Staubli VAL3: onStart.pgx

program onStart()
  local num i
begin
  // logMsg
  logMsg("[KERNEL] INTERFACE:PAGE Edit trajectory")
  // disable the filter
  if saveData:mode<2
    saveData:sTrajFilter=""
  endIf
  // check it
  if saveData:sTrajType[nType]!=saveData:sTrajTypeUsing
    for i=0 to size(saveData:sTrajType)-1
      // scan
      if saveData:sTrajTypeUsing==saveData:sTrajType[i]
        nType=i
        i=size(saveData:sTrajType)-1
      endIf
    endFor
  endIf
  // reset the Key pressure
  call use:nullKey(nKey)
  // define the select traj
  call defineTraj()
  // clean the userMenu
  call cleanUserMenu()
  // define the list
  call buildList()
end
